{attribute 'call_after_init'}
{attribute 'reflection'}
FUNCTION_BLOCK PUBLIC BoolOut EXTENDS SymbolPathStorage IMPLEMENTS I_StepCondition
VAR_INPUT
END_VAR
VAR_OUTPUT
END_VAR
VAR
	{attribute 'instance-path'}  
	{attribute 'no_init'} 
	sPath : T_MaxString;
	bValue AT%Q* : BOOL;
	sInitPath : T_MaxString;

END_VAR

{attribute 'call_after_init'}
METHOD PRIVATE CallAfterInit : BOOL
IF uiPathCounter <= cMaxPaths 
THEN
	//Delete the part of the path which contains solution and project name 	
	sInitPath := DELETE(sPath,FIND(sPath,'.'),1);
	sInitPath := DELETE(sInitPath,FIND(sInitPath,'.'),1);
	sInitPath := CONCAT(sInitPath,'.bValue');
	aPaths[uiPathCounter] := sInitPath;
	uiPathCounter := uiPathCounter + 1;
END_IF
END_METHOD


PROPERTY getValue : BOOL
GET
getValue := bValue;
END_GET
END_PROPERTY


PROPERTY setValue : BOOL
SET
bValue := setValue;
END_SET
END_PROPERTY

END_FUNCTION_BLOCK

(* stored: Version 1.1.0.1, ProductVersion 3.1.4024.2
   POU BoolOut: Id {c33c3c8d-1af1-4fe2-9050-6b44e83ade36}, SpecialFunc None
   Method CallAfterInit: Id {400f6a9f-5fff-43fb-8d37-a345e228c015}
   Property getValue: Id {4e500a82-3cd9-45de-9d49-40b45ccd2d96}
   Get Get: Id {baa3866a-09e3-4c48-9aa7-022a2e4a6248}
   Property setValue: Id {708f6d83-f6e5-4439-a3bc-c4ffe722bfbd}
   Set Set: Id {6d3123a9-2116-4846-8e6a-ce53eb573339} *)
